FUNCTION_BLOCK PUBLIC FB_DevAnalogInput EXTENDS FB_DevBase
VAR_INPUT
	bCmdSimulate	: BOOL 	:= FALSE ;// Simulate sensor Input 
	fSimValue		: INT	:= 0 ;// Simulated sensor state
END_VAR
VAR_OUTPUT
	fValue	: LREAL := 0 ; // Input value from hardware (converted to LREAL)
END_VAR
VAR
	nLimitMin		: INT := Utilities_Library.GVL_FixedValues.nINTMINVALUE ; // Initial value is set to integer minimum value for use with normal def analog inputs 
	nLimitMax 		: INT := Utilities_Library.GVL_FixedValues.nINTMAXVALUE	; // Initial value is set to integer minimum value for use with high def analog inputs
	inHwInput AT%I* : INT ; // Hardware connection
END_VAR

// Set device type
eDevType := E_Devices.AnalogSensor ;

// Call base function
SUPER^(refFbFault := refFbFault);

// set feedback
ExecSetFeedback();

METHOD ExecSetFeedback : BOOL
VAR_INPUT
END_VAR
IF bCmdSimulate THEN 
	fValue := int_to_lreal(fSimValue) ;
ELSE
	fValue := INT_TO_LREAL(inHwInput);
END_IF
END_METHOD

METHOD PUBLIC Init : BOOL
VAR_INPUT
	// Location data for messages  
	nId			: UDINT ; // Identification number of object
	nParentId	: UDINT ; // Id of higher level If aplicable (0 = no parent)
END_VAR
// ====== Calculate device id =====
	ExecIdentifyDevice(nId,nParentId);

// ====== Set feedback ======
	bInitOk := true ;
END_METHOD

END_FUNCTION_BLOCK

(* stored: Version 1.1.0.1, ProductVersion 3.1.4024.5
   POU FB_DevAnalogInput: Id {438fca26-964b-0408-10a5-3e8ee84a0164}, SpecialFunc None
   Method ExecSetFeedback: Id {7a115a3e-3411-01c5-2bf8-56b6258af2f3}
   Method Init: Id {3357007e-f480-0c2c-080e-7ce021956725} *)
